FUNCTION_BLOCK OutputDecompressor (* Basic Function Block Type *)
  (* Standard: 61499-2 *)
  (* Version 0.0, 11/2/2016, Dmitry, nxtControl GmbH, Template *)
  PACKAGE Main;
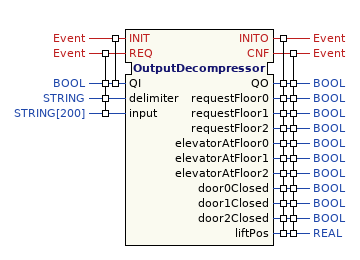
  EVENT_INPUT
    INIT WITH QI; (* Initialization Request *)
    REQ WITH QI, delimiter, input; (* Normal Execution Request *)
  END_EVENT
  EVENT_OUTPUT
    INITO WITH QO, requestFloor0, requestFloor1, requestFloor2, elevatorAtFloor0, elevatorAtFloor1, elevatorAtFloor2, door0Closed, door1Closed, door2Closed, liftPos; (* Initialization Confirm *)
    CNF WITH QO, requestFloor0, requestFloor1, requestFloor2, elevatorAtFloor0, elevatorAtFloor1, elevatorAtFloor2, door0Closed, door1Closed, door2Closed, liftPos; (* Execution Confirmation *)
  END_EVENT
  VAR_INPUT
    QI : BOOL; (* Input event qualifier *)
    delimiter : STRING;
    input : STRING[200];
  END_VAR
  VAR_OUTPUT
    QO : BOOL; (* Output event qualifier *)
    requestFloor0 : BOOL;
    requestFloor1 : BOOL;
    requestFloor2 : BOOL;
    elevatorAtFloor0 : BOOL;
    elevatorAtFloor1 : BOOL;
    elevatorAtFloor2 : BOOL;
    door0Closed : BOOL;
    door1Closed : BOOL;
    door2Closed : BOOL;
    liftPos : REAL;
  END_VAR
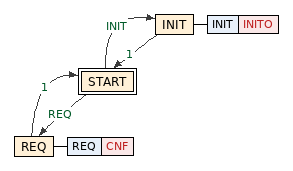
  EC_STATES
    START; (* Initial State *)
    INIT : INIT -> INITO; (* Initialization *)
    REQ : REQ -> CNF; (* Normal execution *)
  END_STATES
  EC_TRANSITIONS
    START TO INIT := INIT;
    INIT TO START := 1;
    START TO REQ := REQ;
    REQ TO START := 1;
  END_TRANSITIONS
  ALGORITHM INIT IN ST: (* Initialization algorithm *)
QO := TRUE;
  END_ALGORITHM
  ALGORITHM REQ IN ST: (* Normally executed algorithm *)
VAR
	length: INT;
	i : INT;
	prev: INT;
	subs : ARRAY[1..18] OF STRING;
	num : INT;
	cur: INT;
END_VAR
length := DINT_TO_INT(LEN(input));
prev := 1;
cur := 1;
FOR i := 1 TO length DO
	IF (MID(input,1,i) = delimiter) THEN
		subs[cur] := MID(input, i - prev, prev);//input.DATA[prev, i-1];
		cur := cur + 1;
		prev := i + 1;
	END_IF;
END_FOR;
(*buttonFloor0 := STRING_TO_BOOL(subs[1]);
buttonFloor1 := STRING_TO_BOOL(subs[2]);
buttonFloor2 := STRING_TO_BOOL(subs[3]);*)
requestFloor0 := STRING_TO_BOOL(subs[1]);
requestFloor1 := STRING_TO_BOOL(subs[2]);
requestFloor2 := STRING_TO_BOOL(subs[3]);
elevatorAtFloor0 := STRING_TO_BOOL(subs[4]);
elevatorAtFloor1 := STRING_TO_BOOL(subs[5]);
elevatorAtFloor2 := STRING_TO_BOOL(subs[6]);
door0Closed := STRING_TO_BOOL(subs[7]);
door1Closed := STRING_TO_BOOL(subs[8]);
door2Closed := STRING_TO_BOOL(subs[9]);
liftPos := STRING_TO_INT(subs[10]);
  END_ALGORITHM
END_FUNCTION_BLOCK
